# EPICS substitutions: db/Beckhoff_7XXX/ecmcELM7222-0010.substitutions
file "ecmcEL72XX_DRV.template"
{
  pattern {CH_ID}
          {01   }
          {02   }
}

file "ecmcEL72XX_ENC.template"
{
  pattern {CH_ID}
          {01   }
          {02   }
}
